GLOBALCONSTANTS DefaultPool_AI_Numeric (* Numeric object pool constants (ID, Scale, Offset, Decimals) *)
  PACKAGE Uebungen::const::UT::AI;
  VAR_GLOBAL CONSTANT
    OutputNumber_c1_N : logiBUS::utils::conversion::phys::NumericObjectPool_S := (u16ObjId := 12001, r32Scale := 1.0, i32Offset := 0, u8Decimals := 0);
    OutputNumber_c9_N : logiBUS::utils::conversion::phys::NumericObjectPool_S := (u16ObjId := 12009, r32Scale := 1.0, i32Offset := 0, u8Decimals := 0);
    OutputNumber_c10_N : logiBUS::utils::conversion::phys::NumericObjectPool_S := (u16ObjId := 12010, r32Scale := 1.0, i32Offset := 0, u8Decimals := 0);
    OutputNumber_c11_N : logiBUS::utils::conversion::phys::NumericObjectPool_S := (u16ObjId := 12011, r32Scale := 1.0, i32Offset := 0, u8Decimals := 0);
    OutputNumber_c12_N : logiBUS::utils::conversion::phys::NumericObjectPool_S := (u16ObjId := 12012, r32Scale := 1.0, i32Offset := 0, u8Decimals := 0);
    OutputNumber_c2_N : logiBUS::utils::conversion::phys::NumericObjectPool_S := (u16ObjId := 12013, r32Scale := 1.0, i32Offset := 0, u8Decimals := 0);
    OutputNumber_c3_N : logiBUS::utils::conversion::phys::NumericObjectPool_S := (u16ObjId := 12014, r32Scale := 1.0, i32Offset := 0, u8Decimals := 0);
    OutputNumber_c4_N : logiBUS::utils::conversion::phys::NumericObjectPool_S := (u16ObjId := 12015, r32Scale := 1.0, i32Offset := 0, u8Decimals := 0);
    OutputNumber_c5_N : logiBUS::utils::conversion::phys::NumericObjectPool_S := (u16ObjId := 12016, r32Scale := 1.0, i32Offset := 0, u8Decimals := 0);
    OutputNumber_c6_N : logiBUS::utils::conversion::phys::NumericObjectPool_S := (u16ObjId := 12017, r32Scale := 1.0, i32Offset := 0, u8Decimals := 0);
    OutputNumber_c7_N : logiBUS::utils::conversion::phys::NumericObjectPool_S := (u16ObjId := 12018, r32Scale := 1.0, i32Offset := 0, u8Decimals := 0);
    OutputNumber_c8_N : logiBUS::utils::conversion::phys::NumericObjectPool_S := (u16ObjId := 12019, r32Scale := 1.0, i32Offset := 0, u8Decimals := 0);
    OutputNumber_Tick_N : logiBUS::utils::conversion::phys::NumericObjectPool_S := (u16ObjId := 12020, r32Scale := 1.0, i32Offset := 0, u8Decimals := 0);
    OutputNumber_AI_I01_RAW_N : logiBUS::utils::conversion::phys::NumericObjectPool_S := (u16ObjId := 12021, r32Scale := 1.0, i32Offset := 0, u8Decimals := 0);
    OutputNumber_AI_I01_PERCENT_N : logiBUS::utils::conversion::phys::NumericObjectPool_S := (u16ObjId := 12022, r32Scale := 0.0244200244, i32Offset := 0, u8Decimals := 1);
    OutputNumber_AI_I02_RAW_N : logiBUS::utils::conversion::phys::NumericObjectPool_S := (u16ObjId := 12023, r32Scale := 1.0, i32Offset := 0, u8Decimals := 0);
    OutputNumber_AI_I02_PERCENT_N : logiBUS::utils::conversion::phys::NumericObjectPool_S := (u16ObjId := 12024, r32Scale := 0.0244200244, i32Offset := 0, u8Decimals := 1);
    OutputNumber_AI_I03_RAW_N : logiBUS::utils::conversion::phys::NumericObjectPool_S := (u16ObjId := 12025, r32Scale := 1.0, i32Offset := 0, u8Decimals := 0);
    OutputNumber_AI_I03_PERCENT_N : logiBUS::utils::conversion::phys::NumericObjectPool_S := (u16ObjId := 12026, r32Scale := 0.0244200244, i32Offset := 0, u8Decimals := 1);
    OutputNumber_AI_I04_RAW_N : logiBUS::utils::conversion::phys::NumericObjectPool_S := (u16ObjId := 12027, r32Scale := 1.0, i32Offset := 0, u8Decimals := 0);
    OutputNumber_AI_I04_PERCENT_N : logiBUS::utils::conversion::phys::NumericObjectPool_S := (u16ObjId := 12028, r32Scale := 0.0244200244, i32Offset := 0, u8Decimals := 1);
    OutputNumber_AI_I05_RAW_N : logiBUS::utils::conversion::phys::NumericObjectPool_S := (u16ObjId := 12029, r32Scale := 1.0, i32Offset := 0, u8Decimals := 0);
    OutputNumber_AI_I05_PERCENT_N : logiBUS::utils::conversion::phys::NumericObjectPool_S := (u16ObjId := 12030, r32Scale := 0.0244200244, i32Offset := 0, u8Decimals := 1);
    OutputNumber_AI_I06_RAW_N : logiBUS::utils::conversion::phys::NumericObjectPool_S := (u16ObjId := 12031, r32Scale := 1.0, i32Offset := 0, u8Decimals := 0);
    OutputNumber_AI_I06_PERCENT_N : logiBUS::utils::conversion::phys::NumericObjectPool_S := (u16ObjId := 12032, r32Scale := 0.0244200244, i32Offset := 0, u8Decimals := 1);
    OutputNumber_AI_I07_RAW_N : logiBUS::utils::conversion::phys::NumericObjectPool_S := (u16ObjId := 12033, r32Scale := 1.0, i32Offset := 0, u8Decimals := 0);
    OutputNumber_AI_I07_PERCENT_N : logiBUS::utils::conversion::phys::NumericObjectPool_S := (u16ObjId := 12034, r32Scale := 0.0244200244, i32Offset := 0, u8Decimals := 1);
    OutputNumber_AI_I08_RAW_N : logiBUS::utils::conversion::phys::NumericObjectPool_S := (u16ObjId := 12035, r32Scale := 1.0, i32Offset := 0, u8Decimals := 0);
    OutputNumber_AI_I08_PERCENT_N : logiBUS::utils::conversion::phys::NumericObjectPool_S := (u16ObjId := 12036, r32Scale := 0.0244200244, i32Offset := 0, u8Decimals := 1);
    NumberVariable_AI_I01_N : logiBUS::utils::conversion::phys::NumericObjectPool_S := (u16ObjId := 21000, r32Scale := 0.0244200244, i32Offset := 0, u8Decimals := 1);
    NumberVariable_AI_I02_N : logiBUS::utils::conversion::phys::NumericObjectPool_S := (u16ObjId := 21001, r32Scale := 0.0244200244, i32Offset := 0, u8Decimals := 1);
    NumberVariable_AI_I03_N : logiBUS::utils::conversion::phys::NumericObjectPool_S := (u16ObjId := 21002, r32Scale := 0.0244200244, i32Offset := 0, u8Decimals := 1);
    NumberVariable_AI_I04_N : logiBUS::utils::conversion::phys::NumericObjectPool_S := (u16ObjId := 21003, r32Scale := 0.0244200244, i32Offset := 0, u8Decimals := 1);
    NumberVariable_AI_I05_N : logiBUS::utils::conversion::phys::NumericObjectPool_S := (u16ObjId := 21004, r32Scale := 0.0244200244, i32Offset := 0, u8Decimals := 1);
    NumberVariable_AI_I06_N : logiBUS::utils::conversion::phys::NumericObjectPool_S := (u16ObjId := 21005, r32Scale := 0.0244200244, i32Offset := 0, u8Decimals := 1);
    NumberVariable_AI_I07_N : logiBUS::utils::conversion::phys::NumericObjectPool_S := (u16ObjId := 21006, r32Scale := 0.0244200244, i32Offset := 0, u8Decimals := 1);
    NumberVariable_AI_I08_N : logiBUS::utils::conversion::phys::NumericObjectPool_S := (u16ObjId := 21007, r32Scale := 0.0244200244, i32Offset := 0, u8Decimals := 1);
  END_VAR
END_GLOBALCONSTANTS
(* other elements stored in the file *)
(* ACHTUNG: 'NumberVariable_AI_I01' wird von mehreren Widgets mit unterschiedlicher Skalierung gebunden - 'OutputNumber_AI_I01_RAW' (scale=1.0 offset=0 decimals=0) vs. 'OutputNumber_AI_I01_PERCENT' (scale=0.0244200244 offset=0 decimals=1). Es gilt die Skalierung mit dem kleinsten |Scale|, alle Widgets muessen dieselbe Skalierung haben. *)
(* ACHTUNG: 'NumberVariable_AI_I02' wird von mehreren Widgets mit unterschiedlicher Skalierung gebunden - 'OutputNumber_AI_I02_RAW' (scale=1.0 offset=0 decimals=0) vs. 'OutputNumber_AI_I02_PERCENT' (scale=0.0244200244 offset=0 decimals=1). Es gilt die Skalierung mit dem kleinsten |Scale|, alle Widgets muessen dieselbe Skalierung haben. *)
(* ACHTUNG: 'NumberVariable_AI_I03' wird von mehreren Widgets mit unterschiedlicher Skalierung gebunden - 'OutputNumber_AI_I03_RAW' (scale=1.0 offset=0 decimals=0) vs. 'OutputNumber_AI_I03_PERCENT' (scale=0.0244200244 offset=0 decimals=1). Es gilt die Skalierung mit dem kleinsten |Scale|, alle Widgets muessen dieselbe Skalierung haben. *)
(* ACHTUNG: 'NumberVariable_AI_I04' wird von mehreren Widgets mit unterschiedlicher Skalierung gebunden - 'OutputNumber_AI_I04_RAW' (scale=1.0 offset=0 decimals=0) vs. 'OutputNumber_AI_I04_PERCENT' (scale=0.0244200244 offset=0 decimals=1). Es gilt die Skalierung mit dem kleinsten |Scale|, alle Widgets muessen dieselbe Skalierung haben. *)
(* ACHTUNG: 'NumberVariable_AI_I05' wird von mehreren Widgets mit unterschiedlicher Skalierung gebunden - 'OutputNumber_AI_I05_RAW' (scale=1.0 offset=0 decimals=0) vs. 'OutputNumber_AI_I05_PERCENT' (scale=0.0244200244 offset=0 decimals=1). Es gilt die Skalierung mit dem kleinsten |Scale|, alle Widgets muessen dieselbe Skalierung haben. *)
(* ACHTUNG: 'NumberVariable_AI_I06' wird von mehreren Widgets mit unterschiedlicher Skalierung gebunden - 'OutputNumber_AI_I06_RAW' (scale=1.0 offset=0 decimals=0) vs. 'OutputNumber_AI_I06_PERCENT' (scale=0.0244200244 offset=0 decimals=1). Es gilt die Skalierung mit dem kleinsten |Scale|, alle Widgets muessen dieselbe Skalierung haben. *)
(* ACHTUNG: 'NumberVariable_AI_I07' wird von mehreren Widgets mit unterschiedlicher Skalierung gebunden - 'OutputNumber_AI_I07_RAW' (scale=1.0 offset=0 decimals=0) vs. 'OutputNumber_AI_I07_PERCENT' (scale=0.0244200244 offset=0 decimals=1). Es gilt die Skalierung mit dem kleinsten |Scale|, alle Widgets muessen dieselbe Skalierung haben. *)
(* ACHTUNG: 'NumberVariable_AI_I08' wird von mehreren Widgets mit unterschiedlicher Skalierung gebunden - 'OutputNumber_AI_I08_RAW' (scale=1.0 offset=0 decimals=0) vs. 'OutputNumber_AI_I08_PERCENT' (scale=0.0244200244 offset=0 decimals=1). Es gilt die Skalierung mit dem kleinsten |Scale|, alle Widgets muessen dieselbe Skalierung haben. *)
